Staubli VAL3: argumentParse.pgx

program argumentParse(num& nBuffer[] (dimensions=1), num nBytes (dimensions=1), num& nArgs[] (dimensions=1), num& nNbArgs (dimensions=1), string& sBuffer (dimensions=1), string& sCommand (dimensions=1))
  local bool bFlag
  local num nIndex
  local num ni
begin
  //convert to string and parse socket data
  sBuffer=""
  //CONVERT TO STRING
  for ni=0 to (nBytes-1) step 1
    sBuffer=sBuffer+chr(nBuffer[ni])
  endFor
  //GET COMMAND NAME
  sCommand=""
  nNbArgs=0
  nIndex=find(sBuffer," ")
  if nIndex==-1
    //command without arguments
    sCommand=sBuffer
  else
    //command with arguments
    sCommand=left(sBuffer,nIndex)
    //GET ARGUMENTS
    //skip space right side characters
    sBuffer=right(sBuffer,nBytes-len(sCommand)-1)
    while (asc(sBuffer,0)==32) and (len(sBuffer)>0)
      sBuffer=right(sBuffer,len(sBuffer)-1)
    endWhile
    //extract arguments
    bFlag=false
    do
      sBuffer=toNum(sBuffer,nArgs[nNbArgs],bFlag)
      nNbArgs=nNbArgs+1
    until (bFlag!=true) or (nNbArgs>8)
    nNbArgs=nNbArgs-1
  endIf
end
